FUNCTION_BLOCK PUBLIC FB_PtpDiagReader
VAR_INPUT
END_VAR
VAR_OUTPUT
	diagInfo: ST_PtpDiag;
END_VAR
VAR
	running: BOOL := FALSE;
	first: BOOL := TRUE;
	netId: T_AmsNetId;
	port: UINT; 
	index: WORD := 16#FA80;
	subIndex: BYTE := 0;
	reader: FB_EcCoESdoReadEx;
	buf: ST_PtpDiag;
	readInterval: TIME := T#1S;
	timer: TON;
	c1: LINT := 0;
	c2: LINT := 0;
	c3: LINT := 0;
	c4: LINT := 0;
END_VAR

// The first time through, get the required ADS parameters.
IF first THEN
	first := FALSE;
	netId := F_CreateAmsNetId(GVL.ptpAdsAddr.netId);
	port := GVL.ptpAdsAddr.port;
	timer(IN:=TRUE, PT:=readInterval);
END_IF

timer();
// If a request is in progress then check for completion.
IF running THEN
	c1 := c1 + 1;
	reader(bExecute:=running);
	IF NOT reader.bBusy THEN
		c2 := c2 + 1;
		diagInfo := buf;
		running := FALSE;
		reader(bExecute:=running);
	END_IF
ELSE
	c3 := c3 + 1;
	IF timer.Q THEN
		timer(IN:=FALSE);
	    running := TRUE;
		timer(IN:=running);
	    reader(sNetId:=netId, nSlaveAddr:=port, nSubIndex:=subIndex, nIndex:=index, pDstBuf:=ADR(buf), cbBufLen:=SIZEOF(buf), bCompleteAccess:=TRUE, bExecute:=running);
	    IF reader.bBusy THEN
		    c4 := c4 + 1;
	    END_IF
	END_IF
END_IF

END_FUNCTION_BLOCK

(* stored: Version 1.1.0.1, ProductVersion 3.1.4022.18
   POU FB_PtpDiagReader: Id {2d2fe6ed-77b1-4d14-9ee0-4b4db2db37c5}, SpecialFunc None *)
